FUNCTION MF_R : real
VAR_INPUT
	x,d,c:REAL;(*a defines the foot of the membership function, AND b defines its shoulder.*)

END_VAR
VAR_OUTPUT
	Error:BOOL;
END_VAR

IF NOT(c=d) AND (c<d) THEN
	IF x>d THEN
		MF_R:=0;
	ELSIF c<=x AND x<=d THEN
		MF_R:=(d-x)/(d-c);
	ELSIF  x<c THEN
		MF_R:=1;
	END_IF
ELSE
	Error:=TRUE;		
END_IF

END_FUNCTION

(* stored: Version 1.1.0.1, ProductVersion 3.1.4024.6
   POU MF_R: Id {3b116fa9-b828-4d7c-b780-c9a1b1fd5e7b}, SpecialFunc None *)
